{attribute 'linkalways'} 
{attribute 'no_explicit_call' := 'This FB is a CLASS and must be accessed using methods or properties'}
{attribute 'enable_dynamic_creation'}
FUNCTION_BLOCK Node_F_VN_BilateralFilter EXTENDS VisionNode
VAR
	ipSrcImage : _ITcVnImage;
    ipDestImage : _ITcVnImage;
    nDiameter : _DINT(1);
    fSigmaColor : _LREAL(10.0);
    fSigmaSpace : _LREAL(10.0);
    hrPrev : _HRESULT(S_OK);
	hresult : _HRESULT(S_OK);
END_VAR

METHOD PUBLIC  Clone : I_Node
VAR
	pNode : POINTER TO Node_F_VN_BilateralFilter;
END_VAR
pNode := __NEW(Node_F_VN_BilateralFilter);
Clone := pNode^;
END_METHOD

METHOD FB_init : BOOL
VAR_INPUT
	bInitRetains : BOOL; // if TRUE, the retain variables are initialized (warm start / cold start)
	bInCopyCode : BOOL;  // if TRUE, the instance afterwards gets moved into the copy code (online change)
END_VAR
AddInput('ipSrcImage', ipSrcImage);
AddParameter('nDiameter', nDiameter);
AddParameter('fSigmaColor', fSigmaColor);
AddParameter('fSigmaSpace', fSigmaSpace);
AddInput('hrPrev', hrPrev);
AddOutput('ipDestImage', ipDestImage);
AddOutput('hresult',hresult);
END_METHOD

METHOD PROTECTED OnExecute
hresult.Value := F_VN_BilateralFilter(
	ipSrcImage:= ipSrcImage.Value,
	ipDestImage:= ipDestImage.Value,
	nDiameter:= nDiameter.Value,
    fSigmaColor := fSigmaColor.Value,
    fSigmaSpace := fSigmaSpace.Value,
	hrPrev:= hrPrev.Value);
END_METHOD

METHOD PUBLIC PreExecutionCheck
VAR_INPUT
	Check : I_PreExecutionChecks;
END_VAR
Check.IsTrue(ipSrcImage.IsValid, 'ipSrcImage must contain an image');
Check.IsTrue((ipSrcImage.HasChannelCount(1) OR ipSrcImage.HasChannelCount(3)), 'ipSrcImage must have 1 or 3 channels');
Check.IsTrue(ipSrcImage.IsPixelDepth(8), 'ipSrcImage must have 8 bit pixel depth');
Check.IsTrue((nDiameter.IsOdd OR nDiameter.Value = 0),'nDiameter must be odd or 0');
Check.IsTrue(fSigmaColor.Value > 0, 'fSigmaColor must be greater than 0');
Check.IsTrue(fSigmaSpace.Value > 0, 'fSigmaSpace must be greater than 0');
END_METHOD

END_FUNCTION_BLOCK

(* stored: Version 1.1.0.1, ProductVersion 3.1.4024.15
   POU Node_F_VN_BilateralFilter: Id {44b7e87b-8473-0131-0405-039e71bf9746}, SpecialFunc None
   Folder Constructor: Id {6e7a4b4e-c64a-034d-1131-ea46e0831b2e}
   Method Clone: Id {76248ecd-a6c3-0334-21ad-ecaf19457610}
   Method FB_init: Id {5fca4477-6e75-0155-35b7-38f860cff209}
   Method OnExecute: Id {0db5b78f-7200-0e18-2da3-809e83715428}
   Method PreExecutionCheck: Id {e274c65d-ed4c-039e-2a5d-e7eacfafaa92} *)
